FUNCTION_BLOCK ValveController
TITLE = 'Valve Controller Function Chart'

// Define inputs
VAR_INPUT
    AutoMode : BOOL;        // Automatic mode switch
    ManualMode : BOOL;      // Manual mode switch
    Interlock : BOOL;       // Interlock input
    AutoOpenCmd : BOOL;     // Valve open pulse command in auto mode
    AutoCloseCmd : BOOL;    // Valve close pulse command in auto mode
    ManualOpenCmd : BOOL;   // Valve open pulse command in manual mode
    ManualCloseCmd : BOOL;  // Valve close pulse command in manual mode
END_VAR

// Define outputs
VAR_OUTPUT
    ValveOpen : BOOL;       // Valve open pulse output
    ValveClose : BOOL;      // Valve close pulse output
    ValveStatus : BOOL;     // Valve status output (true if open, false if closed)
    InterlockStatus : BOOL; // Interlock status output (true if interlocked)
    ValveInManual : BOOL;   // Manual mode status output (true if active)
    ValveInAuto : BOOL;     // Automatic mode status output (true if active)
END_VAR
// Main program
BEGIN
    IF AutoMode THEN
        ValveInAuto := TRUE;
        ValveInManual := FALSE;
    ELSIF ManualMode THEN
        ValveInAuto := FALSE;
        ValveInManual := TRUE;
    END_IF;
    IF Interlock THEN
        // Stop valve movement if interlock is active
        ValveOpen := FALSE;
        ValveClose := FALSE;
        ValveStatus := FALSE;
        InterlockStatus := TRUE;
    ELSIF ValveInAuto THEN // Ventilen er i automode
        IF AutoOpenCmd THEN
            // Open valve in auto mode
            ValveOpen := TRUE;
            ValveClose := FALSE;
            ValveStatus := TRUE;
            InterlockStatus := FALSE;
        ELSIF AutoCloseCmd THEN
            // Close valve in auto mode
            ValveOpen := FALSE;
            ValveClose := TRUE;
            ValveStatus := FALSE;
            InterlockStatus := FALSE;
        END_IF;
    ELSIF ValveInManual THEN
        IF ManualOpenCmd THEN
            // Open valve in manual mode
            ValveOpen := TRUE;
            ValveClose := FALSE;
            ValveStatus := TRUE;
            InterlockStatus := FALSE;
        ELSIF ManualCloseCmd THEN
            // Close valve in manual mode
            ValveOpen := FALSE;
            ValveClose := TRUE;
            ValveStatus := FALSE;
            InterlockStatus := FALSE;
        END_IF;
    END_IF;
END_FUNCTION_BLOCK
